{attribute addProperty BoxType "EM7004-0000-9996"}
{attribute addProperty Id "OutputAT %Q*ARRAY[0 ..15] OF BOOL128160"}
{attribute addProperty CRC "1232143113"}
{attribute addProperty SizeInBites "128"}
{attribute addProperty SizeInBytes "16"}
TYPE DO_Outputs_BF554446 :
STRUCT
	{attribute addProperty Name "Output"}
	Output AT %Q* : ARRAY[0 ..15] OF BOOL;
END_STRUCT
END_TYPE

(* stored: Version 1.2.0.0, ProductVersion 3.1.4024.9
   DUT DO_Outputs_BF554446: Id {43d4c9e2-c0d1-4b4a-b1f0-df6214c4a31d} *)
